PROGRAM MAIN
VAR
	fbLogger:			Tc3_Event.FB_LoggerManager;
	fbHmiLogger:		Tc3_Event.FB_HmiLogger;
	fbFileLogger:		Tc3_Event.FB_FileLogger;
	fbTcLogger:			Tc3_Event.FB_TcLogger;
	fbTest:				FB_TestSlow;
  	exception:			__SYSTEM.ExceptionCode;	
	bReset: BOOL;
END_VAR

__TRY
	IF exception = __SYSTEM.ExceptionCode.RTSEXCPT_NOEXCEPTION THEN
		fbLogger.M_Add(fbHmiLogger);
		fbLogger.M_Add(fbFileLogger);
		fbLogger.M_Add(fbTcLogger);
			
		fbHmiLogger();
		fbFileLogger.sPathName:= 'C:\temp\log.txt';
		fbFileLogger();
		fbTcLogger();
		
		IF bReset THEN
			fbLogger.M_Reset();
		END_IF
		
		
		
		fbTest.P_Event.P_Logger:= fbLogger;
		
		fbTest();		
	END_IF

__CATCH(exception)

__ENDTRY

END_PROGRAM

(* stored: Version 1.1.0.1
   POU MAIN: Id {19c7fd4e-92ee-4c48-b527-6576c9627f78}, SpecialFunc None *)
